FUNCTION_BLOCK FB_MyQ_REAL_OOP_v2
VAR CONSTANT
	QUEUESIZE: UDINT := 10;
END_VAR
VAR
	HoldQueue: ARRAY[1..QUEUESIZE] OF REAL;
	ProcessQueue: ARRAY[1..QUEUESIZE] OF REAL;
	Elements: UDINT;
END_VAR

METHOD M_Copy : ARRAY[1..QUEUESIZE] OF REAL
MEMCPY(ADR(M_Copy[1]), ADR(ProcessQueue[1]), SIZEOF(M_Copy));
END_METHOD

METHOD M_Insert : BOOL
VAR_INPUT
	NewValue: REAL;
END_VAR
IF Elements < QUEUESIZE THEN
	Elements := Elements + 1;
	ProcessQueue[Elements]:= NewValue;
ELSE
	Elements := QUEUESIZE;	
	MEMCPY(ADR(HoldQueue[1]), ADR(ProcessQueue[1]), SIZEOF(HoldQueue)); 
	MEMCPY(ADR(ProcessQueue[1]), ADR(HoldQueue[2]), SIZEOF(ProcessQueue)-SIZEOF(REAL));
	MEMSET(ADR(ProcessQueue[Elements]), 0, SIZEOF(REAL));
	ProcessQueue[Elements]:= NewValue;
END_IF
END_METHOD

METHOD M_Peek : REAL
IF Elements > 0 THEN
	M_Peek := ProcessQueue[1];
END_IF
END_METHOD

METHOD M_Remove : REAL
IF Elements > 0 THEN
	M_Remove := ProcessQueue[1];
	MEMCPY(ADR(HoldQueue[1]), ADR(ProcessQueue[1]), SIZEOF(HoldQueue)); 
	MEMCPY(ADR(ProcessQueue[1]), ADR(HoldQueue[2]), SIZEOF(ProcessQueue)-SIZEOF(REAL));
	MEMSET(ADR(ProcessQueue[Elements]), 0, SIZEOF(REAL));
	Elements := Elements - 1;
END_IF
END_METHOD

METHOD M_Reset : BOOL
MEMSET(ADR(HoldQueue[1]), 0, SIZEOF(HoldQueue));
MEMSET(ADR(ProcessQueue[1]), 0, SIZEOF(ProcessQueue));	
Elements := 0;
END_METHOD

PROPERTY P_Count : UDINT
GET
P_Count:=Elements;
END_GET
END_PROPERTY

PROPERTY P_FIFOSize : UDINT
GET
P_FIFOSize:=QUEUESIZE;
END_GET
END_PROPERTY

END_FUNCTION_BLOCK

(* stored: Version 1.1.0.1, ProductVersion 3.1.4024.3
   POU FB_MyQ_REAL_OOP_v2: Id {48115785-36c3-0733-1ce3-db6e2fcb4227}, SpecialFunc None
   Method M_Copy: Id {978fa762-a161-02fe-108f-f6bafdc31aaf}
   Method M_Insert: Id {ad20217e-4848-0d32-37a5-cb74032d2370}
   Method M_Peek: Id {e6614b49-a211-0974-0057-c9cc0775cfcd}
   Method M_Remove: Id {747d87a7-b45f-0031-1c98-cfbff0e71bcf}
   Method M_Reset: Id {7dfe5407-945e-0527-3df7-4f4793bfe8ae}
   Property P_Count: Id {90c80285-a92f-0bc1-1d0a-2f7e1829662d}
   Get Get: Id {a34e4d9d-ef80-0b59-22da-d31801e0689e}
   Property P_FIFOSize: Id {76cade04-bf17-05ac-1399-eee8d044752d}
   Get Get: Id {963052b7-ca47-0040-0099-73793c91764e} *)
